// TIA Portal project "Sıcaklik Sensoru" (V15.1)

(* hardware
DEVICE "PC-System_1"  SIMATIC PC station
   slot 0: "SIMATIC PC station"  Rail  SIMATIC PC-Station  V1.0
      slot 125: "Stationmanager"  Station_Manager  V6.0.4
   slot 1: "HMI_RT_1"  WinCC RT Advanced  6AV2 104-0xxxx-xxxx  15.1.0.0
      slot 33792: "Host interface"  Host interface
   slot 2: "IE general_1"  IE General  IE_CP  V8.2.0
DEVICE "S7-1200 station_1"  S7-1200 Station
   slot 0: "Rack_0"  S7-1200 Rack  Rack  V1.0
   slot 1: "PLC_1"  CPU 1212C DC/DC/DC  6ES7 212-1AE40-0XB0  V4.1
*)

// ===== PLC "PLC_1"  CPU 1212C DC/DC/DC =====

VAR_GLOBAL   // PLC tag table "Default tag table"
   "stop" AT %M5.0 : Bool;
   "start" AT %M5.1 : Bool;
   "sistem_devrede" AT %M5.2 : Bool;
   "sicaklık_sensoru" AT %MW5 : UInt;
   "sicaklik_akfif" AT %M5.3 : Bool;
END_VAR

ORGANIZATION_BLOCK "Main"   // OB1, LAD, ProgramCycle
TITLE = "Main Program Sweep (Cycle)"
{ S7_Optimized_Access := 'TRUE' }
VERSION : 0.1
   VAR_INPUT
      Initial_Call : Bool;   // Initial call of this OB
      Remanence : Bool;   // =True, if remanent data are available
   END_VAR
BEGIN

REGION Network 1
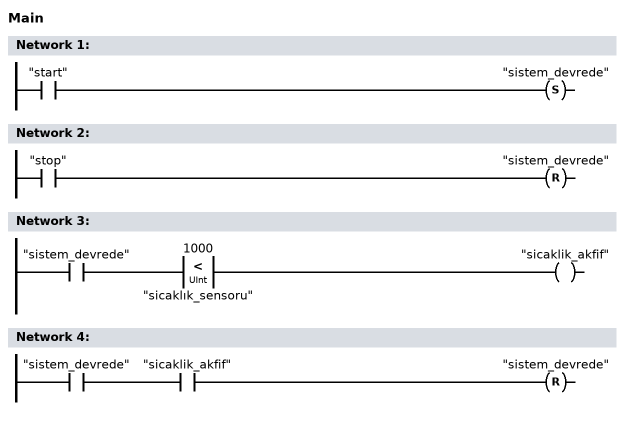
   RUNG wire#powerrail
      Contact( "start" )
      S_Coil( "sistem_devrede" )
   END_RUNG
   // the same network as SCL:
   IF "start" THEN "sistem_devrede" := TRUE; END_IF;
END_REGION

REGION Network 2
   RUNG wire#powerrail
      Contact( "stop" )
      R_Coil( "sistem_devrede" )
   END_RUNG
   // the same network as SCL:
   IF "stop" THEN "sistem_devrede" := FALSE; END_IF;
END_REGION

REGION Network 3
   RUNG wire#powerrail
      Contact( "sistem_devrede" )
      { S7_Templates := "SrcType := UInt" } LT_Contact(in1 := 1000, in2 := "sicaklık_sensoru")
      Coil( "sicaklik_akfif" )
   END_RUNG
   // the same network as SCL:
   "sicaklik_akfif" := "sistem_devrede" AND (1000 < "sicaklık_sensoru");
END_REGION

REGION Network 4
   RUNG wire#powerrail
      Contact( "sistem_devrede" )
      Contact( "sicaklik_akfif" )
      R_Coil( "sistem_devrede" )
   END_RUNG
   // the same network as SCL:
   IF "sistem_devrede" AND "sicaklik_akfif" THEN "sistem_devrede" := FALSE; END_IF;
END_REGION
END_ORGANIZATION_BLOCK

(* ===== HMI "HMI_RT_1" =====
system functions are stored by id; their names below are inferred from use
connection "HMI_Connection_1": ETHERNET, S7_1200_OMS

HMI tags "hmi_tags"
   "HMI_stop" : Bool = PLC stop AT %M5.0, 100 ms
   "HMI_start" : Bool = PLC start AT %M5.1, 100 ms
   "HMI_sensor" : UInt = PLC sicaklık_sensoru AT %MW5, 100 ms
   "HMI_MEMO" : Bool = PLC sicaklik_akfif AT %M5.3, 100 ms

screen "ana_ekran" 1024x768
   Button "Button_1" at 194,189 size 96x34; TextOff 'START'
      on Press: SetBit("HMI_start")
      on Release: ResetBit("HMI_start")
   Button "Button_2" at 194,259 size 96x32; TextOff 'STOPP'
      on Release: ResetBit("HMI_stop")
      on Press: SetBit("HMI_stop")
   Gauge "Gauge_1" at 424,120 size 226x226; CaptionText 'SIMATIC'; UnitText 'Unit'
      ProcessValue <- "HMI_sensor"
   Circle "Circle_1" at 776,168 size 97x97
      Appearance <- "HMI_MEMO"
*)